ABB RobotStudio station: test.rspag

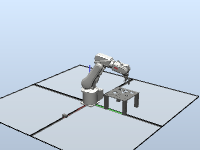
--- station ---
Station test1 (saved by RobotStudio 6.5.7392.129)
Controller System1
  mechanical unit ROB_1: IRB120_3_58__01, 6 joints, base frame (0, 0, 0) mm
Layout (positions relative to the parent item):
  - IRB120_3_58__01 [mechanism, from Robots\IRB120_3_58_G_01.rslib] at (0, 0, 0) mm; joint values [1.7778, 0.5772, -0.3342, 0, 1.3278, 0.207] (rad or m)
  - SmartComponent_1 [smart component] at (-93.97, 447.54, 439.52) mm, rotated rx 180 ry 0 rz -90 deg
      signals: DI GET, DO FINISH
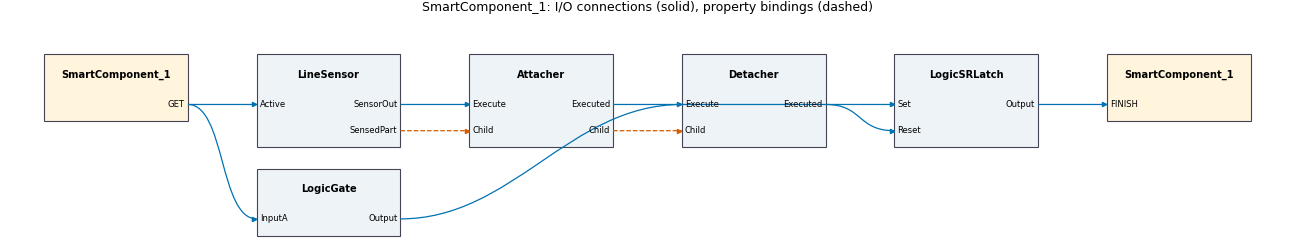
      connections:
        SmartComponent_1.GET -> LineSensor.Active
        SmartComponent_1.GET -> LogicGate.InputA
        LineSensor.SensorOut -> Attacher.Execute
        LogicGate.Output -> Detacher.Execute
        Attacher.Executed -> LogicSRLatch.Set
        Detacher.Executed -> LogicSRLatch.Reset
        LogicSRLatch.Output -> SmartComponent_1.FINISH
        Attacher.Child => Detacher.Child
        LineSensor.SensedPart => Attacher.Child
    - My_Mechanism  [mechanism] at (0, 0, 0) mm; joint values [0.01] (rad or m)
        TCP tool1 at (15.5, 0, 69.3) mm
        TCP tool2 at (-22.5, 0, 83.55) mm
        TCP tool3 at (-22.5, 0, 160.55) mm
        links: L1, L2
    - Attacher [smart component, from Components\Attacher.rslib]
        properties: Parent=SmartComponent_1; Flange=0; Child=TCP-练习笔; Mount=false; Offset=[0.461455780029297 0.0299996566772461 0.0300000019073486]; Orientation=[0 0 0]
    - Detacher [smart component, from Components\Detacher.rslib]
        properties: Child=TCP-练习笔; KeepPosition=true
    - LogicGate [smart component, from Components\LogicGate.rslib]
        properties: Operator=NOT; Delay=0
    - LogicSRLatch [smart component, from Components\LogicSRLatch.rslib]
    - LineSensor [smart component, from Components\LineSensor.rslib] at (-22.5, 0, 81.55) mm
        properties: Start=[0 0 0]; End=[0 0 0.0125]; Radius=0.005; SensedPart=TCP-练习笔; SensedPoint=[-0.0939664688110352 0.470044921875 0.205976928710938]
      - _sensorPart_ [part]
  - 部件_1 [part] at (0, 0, 0) mm
  - TCP_Table [part]
  - TCP-练习笔 [part] at (0, 0, 0) mm
  - 框架_1 [frame] at (15.5, 0, 69.3) mm
  - 框架_2 [frame] at (-22.5, 0, 83.55) mm
  - 框架_3 [frame] at (-22.5, 0, 160.55) mm
Attachment: SmartComponent_1 is attached to IRB120_3_58__01 / Link6
Attachment: LineSensor is attached to My_Mechanism  / L1
EventTableEntry 1008: Group=, Trigger=DO_007 1009, Actions=[EventTableActionMechanicalPose 1010], Comment=, ActivationMode=2, Cyclic=false
EventTableTriggerIO 1009: IOValue=[1], IRC5Controller=? -1, Operator=0, SignalSource=System1 515
EventTableActionMechanicalPose 1010: VirtualSignal=, Mechanism=My_Mechanism  994, ToPoseName=SyncPosition, VirtualSignalValue=[1]
EventTableEntry 1011: Group=, Trigger=DO_007 1012, Actions=[EventTableActionMechanicalPose 1013], Comment=, ActivationMode=2, Cyclic=false
EventTableTriggerIO 1012: IOValue=[0], IRC5Controller=? -1, Operator=0, SignalSource=System1 515
EventTableActionMechanicalPose 1013: VirtualSignal=, Mechanism=My_Mechanism  994, ToPoseName=HomePosition, VirtualSignalValue=[1]
Station logic (signal -> signal, property => property):
  System1.DO_007 -> SmartComponent_1.GET
Targets, tools, work objects and paths stored in the station and not in the controller backup, written as RAPID:
! task T_ROB1
MODULE CalibData
  PERS tooldata tool1:=[TRUE,[[15.5,0,69.3],[1,0,0,0]],[1,[0,0,1],[1,0,0,0],0,0,0]];
  PERS tooldata tool2:=[TRUE,[[-22.5,0,83.548],[1,0,0,0]],[1,[0,0,1],[1,0,0,0],0,0,0]];
  PERS tooldata tool3:=[TRUE,[[-22.5,0,160.548],[1,0,0,0]],[1,[0,0,1],[1,0,0,0],0,0,0]];
ENDMODULE


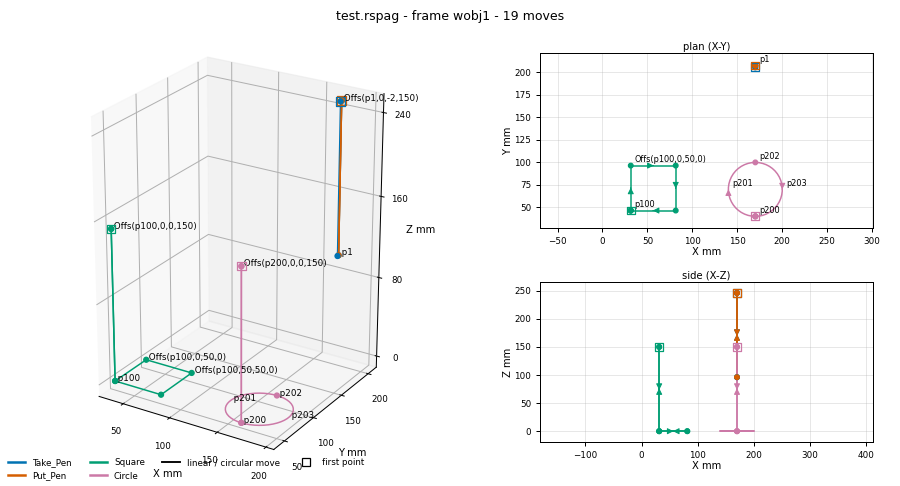
[picture p0: tool path of test.rspag in frame wobj1, 19 of 21 moves have a stored position in this frame; points joined in program order, loops and branches not executed]
--- Backups/System1/RAPID/TASK1/PROGMOD/Module1.mod ---
MODULE Module1
	CONST robtarget p1:=[[169.95,207.74,96.16],[1.07405E-07,-0.707107,0.707107,1.06202E-07],[1,-1,0,0],[9E+09,9E+09,9E+09,9E+09,9E+09,9E+09]];
	CONST robtarget p11:=[[637.92,-239.80,436.64],[0.707107,-8.49626E-15,0.707107,8.12824E-15],[0,0,-1,0],[9E+09,9E+09,9E+09,9E+09,9E+09,9E+09]];
	CONST robtarget p100:=[[31.46,46.46,0.00],[8.96457E-08,3.91016E-08,-1,-2.50508E-07],[1,-1,0,0],[9E+09,9E+09,9E+09,9E+09,9E+09,9E+09]];
	CONST robtarget p110:=[[169.95,230.24,-64.39],[3.22421E-08,2.34657E-09,-1,-1.82593E-07],[1,-1,0,0],[9E+09,9E+09,9E+09,9E+09,9E+09,9E+09]];
	CONST robtarget p200:=[[170.00,40.00,0.00],[5.80683E-08,-2.51812E-07,-1,-2.43058E-07],[1,-1,0,0],[9E+09,9E+09,9E+09,9E+09,9E+09,9E+09]];
	CONST robtarget p220:=[[31.46,46.46,0.00],[8.96457E-08,3.91016E-08,-1,-2.50508E-07],[1,-1,0,0],[9E+09,9E+09,9E+09,9E+09,9E+09,9E+09]];
	CONST robtarget p210:=[[31.46,46.46,0.00],[8.96457E-08,3.91016E-08,-1,-2.50508E-07],[1,-1,0,0],[9E+09,9E+09,9E+09,9E+09,9E+09,9E+09]];
	CONST robtarget p201:=[[140.00,70.00,-0.00],[7.39694E-08,9.4367E-08,-1,-1.19943E-07],[1,0,0,0],[9E+09,9E+09,9E+09,9E+09,9E+09,9E+09]];
	CONST robtarget p202:=[[170.00,100.00,0.00],[1.85824E-07,5.90141E-07,-1,-1.50034E-07],[1,0,0,0],[9E+09,9E+09,9E+09,9E+09,9E+09,9E+09]];
	CONST robtarget p203:=[[200.00,70.00,-0.00],[7.66924E-08,6.83809E-07,-1,-1.34942E-07],[1,0,0,0],[9E+09,9E+09,9E+09,9E+09,9E+09,9E+09]];
	PROC main()
		Initialize;
		Take_Pen;
		Square;
		Circle;
		Put_Pen;
	ENDPROC
	PROC Initialize()
		AccSet 100, 100;
		VelSet 100, 300;
		MoveAbsJ [[0,0,0,0,0,0],[9E+09,9E+09,9E+09,9E+09,9E+09,9E+09]]\NoEOffs, v100, z50, tool0\WObj:=wobj0;
		Reset DO_007;
		MoveAbsJ [[90,-1.21927E-12,-8.32302E-13,1.21817E-18,90,-2.98212E-14],[9E+09,9E+09,9E+09,9E+09,9E+09,9E+09]]\NoEOffs, v100, z50, tool0;
	ENDPROC
	PROC Take_Pen()
		MoveJ Offs(p1,0,-2,150), v100, z50, tool0\WObj:=wobj1;
		MoveL Offs(p1,0,-2,0), v50, fine, tool0\WObj:=wobj1;
		MoveL p1, v50, fine, tool0\WObj:=wobj1;
		Set DO_007;
		WaitTime 1;
		MoveL Offs(p1,0,0,150), v100, z50, tool0\WObj:=wobj1;
	ENDPROC
	PROC Put_Pen()
		MoveJ Offs(p1,0,0,150), v100, z50, tool0\WObj:=wobj1;
		MoveL p1, v50, fine, tool0\WObj:=wobj1;
		Reset DO_007;
		WaitTime 1;
		MoveL Offs(p1,0,0,150), v100, z50, tool0\WObj:=wobj1;
	ENDPROC
	PROC Square()
		MoveJ Offs(p100,0,0,150), v100, z50, tool_pen\WObj:=wobj1;
		MoveL p100, v50, z50, tool_pen\WObj:=wobj1;
		MoveL Offs(p100,0,50,0), v100, z50, tool_pen\WObj:=wobj1;
		MoveL Offs(p100,50,50,0), v100, z50, tool_pen\WObj:=wobj1;
		MoveL Offs(p100,50,0,0), v100, z50, tool_pen\WObj:=wobj1;
		MoveL p100, v100, z50, tool_pen\WObj:=wobj1;
		MoveL Offs(p100,0,0,150), v100, z50, tool_pen\WObj:=wobj1;
	ENDPROC
	PROC Circle()
		MoveJ Offs(p200,0,0,150), v100, z50, tool_pen\WObj:=wobj1;
		MoveL p200, v50, z50, tool_pen\WObj:=wobj1;
		MoveC p201, p202, v100, z10, tool_pen\WObj:=wobj1;
		MoveC p203, p200, v100, z10, tool_pen\WObj:=wobj1;
		MoveL Offs(p200,0,0,150), v100, z50, tool_pen\WObj:=wobj1;
	ENDPROC

ENDMODULE

--- Backups/System1/RAPID/TASK1/SYSMOD/LINKEDM.sys ---
%%%
  VERSION:1
  LANGUAGE:ENGLISH
%%%

MODULE LINKEDM (SYSMODULE)

! FOLLOWER
!     Name of electronically linked follower axis used by operator at teach pendent.
      PERS string l_f_axis_name{5}       :=  ["",  "", "", "", ""];

!     Name of the mechanical unit for follower axis.
      PERS string l_f_mecunt_n{5}  :=  ["", "", "", "", ""];

!     Linked follower axis number in the mechanical unit (first axis in mech. unit is number 1).
      PERS num l_f_axis_no{5}      :=  [0,          0,   0,  0,  0];

! MASTER
!     Name of the mechanical unit for linked master axis.
      PERS string l_m_mecunt_n{5} :=  ["", "", "", "", ""];

!     Linked master axis number in the mechanical unit (first axis in mech. unit is number 1).
!     See axis number table in documentation for different master mechanical units.
      PERS num l_m_axis_no{5}     :=  [0,  0,  0,  0,  0];

! POSITION OFFSET
!     The increase of the allowed offset position between the master and follower
!     positions, used when starting AUTO mode. As soon as the offset is decreased
!     the old configurated parameter is used.
!     Example: 3 => the configurated value of allowed offset is increased 3 times.
      PERS num offset_ratio{5}       :=  [10,  10,   10,  10,  10];

! SPEED RATIO
!     Speed_ratio used in AUTO and JOG modes [ very_slow   slow    normal    fast]
!     Value 1 = max allowed manual speed.
      CONST num speed_ratio {20}      := [0.01, 0.01, 0.01, 0.01, 0.01,
                                          0.05, 0.05, 0.05, 0.05, 0.05,
                                          0.20, 0.20, 0.20, 0.20, 0.20,
                                          1.00, 1.00, 1.00, 1.00, 1.00];

! STEP SIZE
!     Displacement position used in JOG mode for each activation of positive or
!     negative movement.                  [very_short    short   normal   long]
!     Unit degees or meter.
      CONST num displacement {20}     := [0.001, 0.001, 0.001, 0.001, 0.001,
                                          0.005, 0.005, 0.005, 0.005, 0.005,
                                          0.020, 0.020, 0.020, 0.020, 0.020,
                                          0.100, 0.100, 0.100, 0.100, 0.100];


!-------------------------------------------------------------
 PROC Linked_m ()
      Linked_m_exe ;
 ENDPROC
ENDMODULE

--- Backups/System1/SYSPAR/EIO.cfg ---
EIO:CFG_1.0:6:1::
#
INDUSTRIAL_NETWORK:

      -Name "DeviceNet" -Label "DeviceNet Master/Slave Network" -Address "2"
#
DEVICENET_DEVICE:

      -Name "d652" -VendorName "ABB Robotics" -ProductName "24 VDC I/O Device"\
      -Label "DSQC 652 24 VDC I/O Device" -Address 10 -ProductCode 26\
      -DeviceType 7 -ConnectionType "COS" -OutputSize 2 -InputSize 2
#
DEVICENET_INTERNAL_DEVICE:

      -Name "DN_Internal_Device" -VendorName "ABB Robotics"\
      -ProductName "DeviceNet Internal Slave Device"
#
EIO_SIGNAL:

      -Name "DO_007" -SignalType "DO" -Device "d652" -DeviceMap "7"
